// TwinCAT 3 PLC project OEF_4
// ProgramVersion: 3.1.4024.0
// libraries:
//   Tc2_BABasic, * (Beckhoff Automation GmbH)
//   Tc2_Standard, * (Beckhoff Automation GmbH)
//   Tc2_System, * (Beckhoff Automation GmbH)
//   Tc3_Module, * (Beckhoff Automation GmbH)
// project tree:
//   / GlobalTextList.TcGTLO, PlcTask.TcTTO, Visualization Manager.TcVMO (not stored)
//   POUs/ MAIN.TcPOU
//   VISUs/ Visualization.TcVIS
// (motion and I/O tree: see PLC project oef_1)
// real-time tasks:
//   TASK PlcTask: cycle T#10ms, priority 20, ADS port 350
//   TASK PlcTask1: cycle T#10ms, priority 21, ADS port 351
//   TASK PlcTask2: cycle T#10ms, priority 22, ADS port 352
//   TASK PlcTask3: cycle T#10ms, priority 23, ADS port 353
//   TASK PlcTask4: cycle T#10ms, priority 24, ADS port 354
// variable links:
//   OEF_4/OEF_4 Instance <-> Device 1 (EtherCAT)/Term 1 (EK1200)/Term 3 (EL2008)
//     PlcTask Outputs/MAIN.Bled1 <-> Channel 1/Output
//     PlcTask Outputs/MAIN.Bled2 <-> Channel 3/Output

CONFIGURATION OEF_4
    RESOURCE PLC ON TwinCAT3
        TASK PlcTask(INTERVAL := T#10ms, PRIORITY := 23);
        PROGRAM MAIN WITH PlcTask : MAIN;
    END_RESOURCE
END_CONFIGURATION

// ---- POUs/MAIN.TcPOU
PROGRAM MAIN
VAR
	Ngevraagedwarden AT %I*: INT := 0;
	Ngemetewarden AT %I*: INT;
	NScale AT %I*: INT := 100;
	Bled1 AT %Q*: BOOL := 0;
	Bled2 AT %q*: BOOL;
END_VAR

Bled1 := (Ngevraagedwarden - 10)<= LREAL_TO_INT (F_Scale(Ngemetewarden, 0,32767,0,NScale))AND LREAL_TO_INT (F_Scale(Ngemetewarden, 0,32767,0,NScale)) <= (Ngevraagedwarden - 10);
Bled2 := NOT Bled1;

END_PROGRAM

// ---- VISUs/Visualization.TcVIS
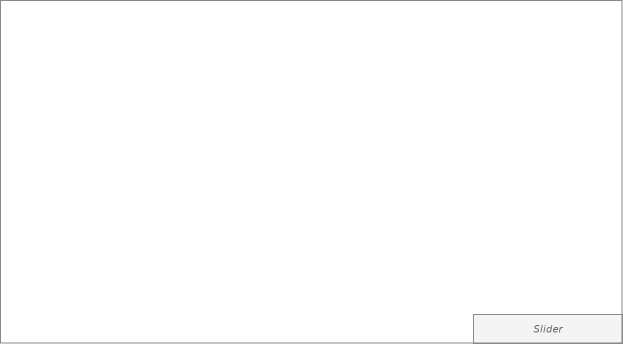
VISUALIZATION Visualization  // 623x344
    Slider (473,314 150x30), variable: MAIN.Ngevraagedwarden, scale 0..100
END_VISUALIZATION
